FUNCTION_BLOCK EffluentActuators (* CAT Function Block Type *)
  (* Standard: 61499-2 *)
  (* Version 0.0, 6/13/2026, Schneider Electric, template *)
  PACKAGE SE.Nereda;
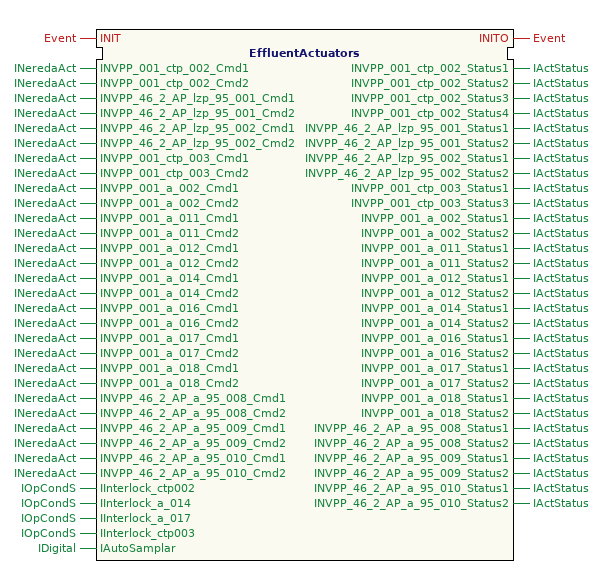
  EVENT_INPUT
    INIT;
  END_EVENT
  EVENT_OUTPUT
    INITO;
  END_EVENT
  SOCKETS
    INVPP_001_ctp_002_Cmd1 : INeredaAct;
    INVPP_001_ctp_002_Cmd2 : INeredaAct;
    INVPP_46_2_AP_lzp_95_001_Cmd1 : INeredaAct;
    INVPP_46_2_AP_lzp_95_001_Cmd2 : INeredaAct;
    INVPP_46_2_AP_lzp_95_002_Cmd1 : INeredaAct;
    INVPP_46_2_AP_lzp_95_002_Cmd2 : INeredaAct;
    INVPP_001_ctp_003_Cmd1 : INeredaAct;
    INVPP_001_ctp_003_Cmd2 : INeredaAct;
    INVPP_001_a_002_Cmd1 : INeredaAct;
    INVPP_001_a_002_Cmd2 : INeredaAct;
    INVPP_001_a_011_Cmd1 : INeredaAct;
    INVPP_001_a_011_Cmd2 : INeredaAct;
    INVPP_001_a_012_Cmd1 : INeredaAct;
    INVPP_001_a_012_Cmd2 : INeredaAct;
    INVPP_001_a_014_Cmd1 : INeredaAct;
    INVPP_001_a_014_Cmd2 : INeredaAct;
    INVPP_001_a_016_Cmd1 : INeredaAct;
    INVPP_001_a_016_Cmd2 : INeredaAct;
    INVPP_001_a_017_Cmd1 : INeredaAct;
    INVPP_001_a_017_Cmd2 : INeredaAct;
    INVPP_001_a_018_Cmd1 : INeredaAct;
    INVPP_001_a_018_Cmd2 : INeredaAct;
    INVPP_46_2_AP_a_95_008_Cmd1 : INeredaAct;
    INVPP_46_2_AP_a_95_008_Cmd2 : INeredaAct;
    INVPP_46_2_AP_a_95_009_Cmd1 : INeredaAct;
    INVPP_46_2_AP_a_95_009_Cmd2 : INeredaAct;
    INVPP_46_2_AP_a_95_010_Cmd1 : INeredaAct;
    INVPP_46_2_AP_a_95_010_Cmd2 : INeredaAct;
    IInterlock_ctp002 : IOpCondS; (* Condition summary chain input from upstream blocks *)
    IInterlock_a_014 : IOpCondS; (* Condition summary chain input from upstream blocks *)
    IInterlock_a_017 : IOpCondS; (* Condition summary chain input from upstream blocks *)
    IInterlock_ctp003 : IOpCondS; (* Condition summary chain input from upstream blocks *)
    IAutoSamplar : IDigital; (* Hardware interface adapter *)
  END_SOCKETS
  PLUGS
    INVPP_001_ctp_002_Status1 : IActStatus;
    INVPP_001_ctp_002_Status2 : IActStatus;
    INVPP_001_ctp_002_Status3 : IActStatus;
    INVPP_001_ctp_002_Status4 : IActStatus;
    INVPP_46_2_AP_lzp_95_001_Status1 : IActStatus;
    INVPP_46_2_AP_lzp_95_001_Status2 : IActStatus;
    INVPP_46_2_AP_lzp_95_002_Status1 : IActStatus;
    INVPP_46_2_AP_lzp_95_002_Status2 : IActStatus;
    INVPP_001_ctp_003_Status1 : IActStatus;
    INVPP_001_ctp_003_Status3 : IActStatus;
    INVPP_001_a_002_Status1 : IActStatus;
    INVPP_001_a_002_Status2 : IActStatus;
    INVPP_001_a_011_Status1 : IActStatus;
    INVPP_001_a_011_Status2 : IActStatus;
    INVPP_001_a_012_Status1 : IActStatus;
    INVPP_001_a_012_Status2 : IActStatus;
    INVPP_001_a_014_Status1 : IActStatus;
    INVPP_001_a_014_Status2 : IActStatus;
    INVPP_001_a_016_Status1 : IActStatus;
    INVPP_001_a_016_Status2 : IActStatus;
    INVPP_001_a_017_Status1 : IActStatus;
    INVPP_001_a_017_Status2 : IActStatus;
    INVPP_001_a_018_Status1 : IActStatus;
    INVPP_001_a_018_Status2 : IActStatus;
    INVPP_46_2_AP_a_95_008_Status1 : IActStatus;
    INVPP_46_2_AP_a_95_008_Status2 : IActStatus;
    INVPP_46_2_AP_a_95_009_Status1 : IActStatus;
    INVPP_46_2_AP_a_95_009_Status2 : IActStatus;
    INVPP_46_2_AP_a_95_010_Status1 : IActStatus;
    INVPP_46_2_AP_a_95_010_Status2 : IActStatus;
  END_PLUGS
  (* 01 - FUNCTIONNAL INPUT INTERFACE *)
  (* 00 - INITIALIZATION *)
  (* 05 - LOGIC *)
  (* 06 - HMI INTERFACE *)
  (* 03 - FIELD INTERFACE *)
  (* 02 - FUNCTIONNAL OUTPUT INTERFACE *)
  (* Actuators Status *)
  (* 04 - CHILDREN *)
  (* 4A - TYPICALS *)
  (* Actuators Command *)
  (* Reset All Actuators *)
  FBS
    ResetAllValves : ResetValvesManager;
    NVPP_001_ctp_002_Status : MultiActStatus;
    NVPP_001_a_002_Status : MultiActStatus;
    NVPP_46_2_AP_lzp_95_001_Status : MultiActStatus;
    NVPP_46_2_AP_lzp_95_002_Status : MultiActStatus;
    NVPP_001_ctp_003_Status : MultiActStatus;
    NVPP_001_ctp_002_Cmd : MultiNeredaCmd;
    NVPP_001_a_002_Cmd : MultiNeredaCmd;
    NVPP_46_2_AP_lzp_95_001_Cmd : MultiNeredaCmd;
    NVPP_001_ctp_003_Cmd : MultiNeredaCmd;
    NVPP_46_2_AP_lzp_95_002_Cmd : MultiNeredaCmd;
    NVPP_001_a_011_Cmd : MultiNeredaCmd;
    NVPP_001_a_012_Cmd : MultiNeredaCmd;
    NVPP_001_a_011_Status : MultiActStatus;
    NVPP_001_a_012_Status : MultiActStatus;
    NVPP_001_a_014_Cmd : MultiNeredaCmd;
    NVPP_001_a_016_Cmd : MultiNeredaCmd;
    NVPP_001_a_014_Status : MultiActStatus;
    NVPP_001_a_016_Status : MultiActStatus;
    NVPP_001_a_017_Cmd : MultiNeredaCmd;
    NVPP_001_a_017_Status : MultiActStatus;
    NVPP_46_2_AP_a_95_008_Cmd : MultiNeredaCmd;
    NVPP_46_2_AP_a_95_009_Cmd : MultiNeredaCmd;
    NVPP_46_2_AP_a_95_008_Status : MultiActStatus;
    NVPP_46_2_AP_a_95_009_Status : MultiActStatus;
    NVPP_46_2_AP_a_95_010_Cmd : MultiNeredaCmd;
    NVPP_46_2_AP_a_95_010_Status : MultiActStatus;
    NVPP_001_a_018_Cmd : MultiNeredaCmd;
    NVPP_001_a_018_Status : MultiActStatus;
    AutoSamplarPulse : dOSignal(Name := '$${PATH}DOut');
  END_FBS
  EVENT_CONNECTIONS
    INIT TO ResetAllValves.INIT;
    ResetAllValves.INITO TO INITO;
  END_CONNECTIONS
  ADAPTER_CONNECTIONS
    INVPP_001_ctp_002_Cmd1 TO NVPP_001_ctp_002_Cmd.F1CE5E5BC0F88348;
    INVPP_001_ctp_002_Cmd2 TO NVPP_001_ctp_002_Cmd.814FBE7646911966;
    INVPP_46_2_AP_lzp_95_001_Cmd1 TO NVPP_46_2_AP_lzp_95_001_Cmd.F1CE5E5BC0F88348;
    INVPP_46_2_AP_lzp_95_001_Cmd2 TO NVPP_46_2_AP_lzp_95_001_Cmd.814FBE7646911966;
    INVPP_46_2_AP_lzp_95_002_Cmd1 TO NVPP_46_2_AP_lzp_95_002_Cmd.F1CE5E5BC0F88348;
    INVPP_46_2_AP_lzp_95_002_Cmd2 TO NVPP_46_2_AP_lzp_95_002_Cmd.814FBE7646911966;
    INVPP_001_ctp_003_Cmd1 TO NVPP_001_ctp_003_Cmd.F1CE5E5BC0F88348;
    INVPP_001_ctp_003_Cmd2 TO NVPP_001_ctp_003_Cmd.814FBE7646911966;
    INVPP_001_a_002_Cmd1 TO NVPP_001_a_002_Cmd.F1CE5E5BC0F88348;
    INVPP_001_a_002_Cmd2 TO NVPP_001_a_002_Cmd.814FBE7646911966;
    INVPP_001_a_011_Cmd1 TO NVPP_001_a_011_Cmd.F1CE5E5BC0F88348;
    INVPP_001_a_011_Cmd2 TO NVPP_001_a_011_Cmd.814FBE7646911966;
    INVPP_001_a_012_Cmd1 TO NVPP_001_a_012_Cmd.F1CE5E5BC0F88348;
    INVPP_001_a_012_Cmd2 TO NVPP_001_a_012_Cmd.814FBE7646911966;
    INVPP_001_a_014_Cmd1 TO NVPP_001_a_014_Cmd.F1CE5E5BC0F88348;
    INVPP_001_a_014_Cmd2 TO NVPP_001_a_014_Cmd.814FBE7646911966;
    INVPP_001_a_016_Cmd1 TO NVPP_001_a_016_Cmd.F1CE5E5BC0F88348;
    INVPP_001_a_016_Cmd2 TO NVPP_001_a_016_Cmd.814FBE7646911966;
    INVPP_001_a_017_Cmd1 TO NVPP_001_a_017_Cmd.F1CE5E5BC0F88348;
    INVPP_001_a_017_Cmd2 TO NVPP_001_a_017_Cmd.814FBE7646911966;
    INVPP_001_a_018_Cmd1 TO NVPP_001_a_018_Cmd.F1CE5E5BC0F88348;
    INVPP_001_a_018_Cmd2 TO NVPP_001_a_018_Cmd.814FBE7646911966;
    INVPP_46_2_AP_a_95_008_Cmd1 TO NVPP_46_2_AP_a_95_008_Cmd.F1CE5E5BC0F88348;
    INVPP_46_2_AP_a_95_008_Cmd2 TO NVPP_46_2_AP_a_95_008_Cmd.814FBE7646911966;
    INVPP_46_2_AP_a_95_009_Cmd1 TO NVPP_46_2_AP_a_95_009_Cmd.F1CE5E5BC0F88348;
    INVPP_46_2_AP_a_95_009_Cmd2 TO NVPP_46_2_AP_a_95_009_Cmd.814FBE7646911966;
    INVPP_46_2_AP_a_95_010_Cmd1 TO NVPP_46_2_AP_a_95_010_Cmd.F1CE5E5BC0F88348;
    INVPP_46_2_AP_a_95_010_Cmd2 TO NVPP_46_2_AP_a_95_010_Cmd.814FBE7646911966;
    NVPP_001_ctp_002_Status.8244952938F4EC92 TO INVPP_001_ctp_002_Status1;
    NVPP_001_ctp_002_Status.3FD61FA75EE1C84B TO INVPP_001_ctp_002_Status2;
    NVPP_001_ctp_002_Status.3A373E4DF127E388 TO INVPP_001_ctp_002_Status3;
    NVPP_001_ctp_002_Status.88456893CB21FD74 TO INVPP_001_ctp_002_Status4;
    NVPP_46_2_AP_lzp_95_001_Status.8244952938F4EC92 TO INVPP_46_2_AP_lzp_95_001_Status1;
    NVPP_46_2_AP_lzp_95_001_Status.3FD61FA75EE1C84B TO INVPP_46_2_AP_lzp_95_001_Status2;
    NVPP_46_2_AP_lzp_95_002_Status.8244952938F4EC92 TO INVPP_46_2_AP_lzp_95_002_Status1;
    NVPP_46_2_AP_lzp_95_002_Status.3FD61FA75EE1C84B TO INVPP_46_2_AP_lzp_95_002_Status2;
    NVPP_001_ctp_003_Status.8244952938F4EC92 TO INVPP_001_ctp_003_Status1;
    NVPP_001_ctp_003_Status.3FD61FA75EE1C84B TO INVPP_001_ctp_003_Status3;
    NVPP_001_a_002_Status.8244952938F4EC92 TO INVPP_001_a_002_Status1;
    NVPP_001_a_002_Status.3FD61FA75EE1C84B TO INVPP_001_a_002_Status2;
    NVPP_001_a_011_Status.8244952938F4EC92 TO INVPP_001_a_011_Status1;
    NVPP_001_a_011_Status.3FD61FA75EE1C84B TO INVPP_001_a_011_Status2;
    NVPP_001_a_012_Status.8244952938F4EC92 TO INVPP_001_a_012_Status1;
    NVPP_001_a_012_Status.3FD61FA75EE1C84B TO INVPP_001_a_012_Status2;
    NVPP_001_a_014_Status.8244952938F4EC92 TO INVPP_001_a_014_Status1;
    NVPP_001_a_014_Status.3FD61FA75EE1C84B TO INVPP_001_a_014_Status2;
    NVPP_001_a_016_Status.8244952938F4EC92 TO INVPP_001_a_016_Status1;
    NVPP_001_a_016_Status.3FD61FA75EE1C84B TO INVPP_001_a_016_Status2;
    NVPP_001_a_017_Status.8244952938F4EC92 TO INVPP_001_a_017_Status1;
    NVPP_001_a_017_Status.3FD61FA75EE1C84B TO INVPP_001_a_017_Status2;
    NVPP_001_a_018_Status.8244952938F4EC92 TO INVPP_001_a_018_Status1;
    NVPP_001_a_018_Status.3FD61FA75EE1C84B TO INVPP_001_a_018_Status2;
    NVPP_46_2_AP_a_95_008_Status.8244952938F4EC92 TO INVPP_46_2_AP_a_95_008_Status1;
    NVPP_46_2_AP_a_95_008_Status.3FD61FA75EE1C84B TO INVPP_46_2_AP_a_95_008_Status2;
    NVPP_46_2_AP_a_95_009_Status.8244952938F4EC92 TO INVPP_46_2_AP_a_95_009_Status1;
    NVPP_46_2_AP_a_95_009_Status.3FD61FA75EE1C84B TO INVPP_46_2_AP_a_95_009_Status2;
    NVPP_46_2_AP_a_95_010_Status.8244952938F4EC92 TO INVPP_46_2_AP_a_95_010_Status1;
    NVPP_46_2_AP_a_95_010_Status.3FD61FA75EE1C84B TO INVPP_46_2_AP_a_95_010_Status2;
    IAutoSamplar TO AutoSamplarPulse.IOut;
  END_CONNECTIONS
END_FUNCTION_BLOCK
